// TIA Portal V15.1 export
// export: Created 2024-06-21T08:40:50.3190684Z, ExportSetting WithDefaults, DisplayName Totally Integrated Automation Portal, DisplayVersion V15.1 Update 5, DisplayName TIA Portal Openness, DisplayVersion V15.1 Update 5, DisplayName SINAMICS Startdrive Advanced, DisplayVersion V15.1, DisplayName G130, G150, S120, S150, SINAMICS MV, S210, DisplayVersion V15.1, DisplayName G110M, G120, G120C, G120D, G120P, DisplayVersion V15.1, DisplayName STEP 7 Professional, DisplayVersion V15.1 Update 5, DisplayName STEP 7 Safety, DisplayVersion V15.1, DisplayName WinCC Professional, DisplayVersion V15.1 Update 5, DisplayName SIMATIC Visualization Architect, DisplayVersion V15.1
DATA_BLOCK "_209230ZS01PNIODiag"   // DB424
{ S7_Optimized_Access := 'FALSE' }
AUTHOR : VCC
VERSION : 0.1
// stored: AutoNumber false, DBAccessibleFromOPCUA true, IsOnlyStoredInLoadMemory false, IsWriteProtectedInAS false
   VAR RETAIN
      "AA_209230AS10-JW60" { ExternalAccessible := 'False'; ExternalVisible := 'False'; ExternalWritable := 'False'} : Bool;   // Profinet device don't exist - ET200sp I/O - Busnode 230AS10 - node 60
      "AA_209230AX01-JW61" { ExternalAccessible := 'False'; ExternalVisible := 'False'; ExternalWritable := 'False'} : Bool;   // Profinet device don't exist - ET200sp I/O - Busnode 230AX01 - node 61
      "AB_209230CA21M4-UE150" { ExternalAccessible := 'False'; ExternalVisible := 'False'; ExternalWritable := 'False'} : Bool;   // Profinet device don't exist - MoviFit - 230CA21M4 - node 150
      "AB_209230CHB21M14-UE151" { ExternalAccessible := 'False'; ExternalVisible := 'False'; ExternalWritable := 'False'} : Bool;   // Profinet device don't exist - MoviFit - 230CHB21M14 - node 151
      "AB_209230CHB22M14-UE152" { ExternalAccessible := 'False'; ExternalVisible := 'False'; ExternalWritable := 'False'} : Bool;   // Profinet device don't exist - MoviFit - 230CHB22M14 - node 152
      "AB_209230CR22M1-UE153" { ExternalAccessible := 'False'; ExternalVisible := 'False'; ExternalWritable := 'False'} : Bool;   // Profinet device don't exist - MoviFit - 230CR22M1 - node 153
      "AA_209230ASD01-JW190" { ExternalAccessible := 'False'; ExternalVisible := 'False'; ExternalWritable := 'False'} : Bool;   // Profinet device don't exist - Euchner Door - 230ASD01 - node 190
      "AA_209230Field-JW223" { ExternalAccessible := 'False'; ExternalVisible := 'False'; ExternalWritable := 'False'} : Bool;   // Profinet device don't exist - Field Switch - Safety Zone 230 - node 223
      "AC_209230AS10-JW60Fault" { ExternalAccessible := 'False'; ExternalVisible := 'False'; ExternalWritable := 'False'} : Bool;   // Faulty profinet device -> For more detail information look for N.A. alarms in the alarmlist - ET200sp I/O - Busnode 230AS10 - node 60
      "AC_209230AX01-JW61Fault" { ExternalAccessible := 'False'; ExternalVisible := 'False'; ExternalWritable := 'False'} : Bool;   // Faulty profinet device -> For more detail information look for N.A. alarms in the alarmlist - ET200sp I/O - Busnode 230AX01 - node 61
      "AC_209230CA21M4-UE150Fault" { ExternalAccessible := 'False'; ExternalVisible := 'False'; ExternalWritable := 'False'} : Bool;   // Faulty profinet device -> For more detail information look for N.A. alarms in the alarmlist - MoviFit - 230CA21M4 - node 150
      "AC_209230CHB21M14-UE151Fault" { ExternalAccessible := 'False'; ExternalVisible := 'False'; ExternalWritable := 'False'} : Bool;   // Faulty profinet device -> For more detail information look for N.A. alarms in the alarmlist - MoviFit - 230CHB21M14 - node 151
      "AC_209230CHB22M14-UE152Fault" { ExternalAccessible := 'False'; ExternalVisible := 'False'; ExternalWritable := 'False'} : Bool;   // Faulty profinet device -> For more detail information look for N.A. alarms in the alarmlist - MoviFit - 230CHB22M14 - node 152
      "AC_209230CR22M1-UE153Fault" { ExternalAccessible := 'False'; ExternalVisible := 'False'; ExternalWritable := 'False'} : Bool;   // Faulty profinet device -> For more detail information look for N.A. alarms in the alarmlist - MoviFit - 230CR22M1 - node 153
      "AC_209230ASD01-JW190Fault" { ExternalAccessible := 'False'; ExternalVisible := 'False'; ExternalWritable := 'False'} : Bool;   // Faulty profinet device -> For more detail information look for N.A. alarms in the alarmlist - Euchner Door - 230ASD01 - node 190
      "AC_209230Field-JW223Fault" { ExternalAccessible := 'False'; ExternalVisible := 'False'; ExternalWritable := 'False'} : Bool;   // Faulty profinet device -> For more detail information look for N.A. alarms in the alarmlist - Field Switch - Safety Zone 230 - node 223
      "209230AS10-JW60AlarmABCondition" { ExternalAccessible := 'False'; ExternalVisible := 'False'; ExternalWritable := 'False'} : Bool;   // Alarm AB condition
      "209230AX01-JW61AlarmABCondition" { ExternalAccessible := 'False'; ExternalVisible := 'False'; ExternalWritable := 'False'} : Bool;   // Alarm AB condition
      "209230CA21M4-UE150AlarmABCondition" { ExternalAccessible := 'False'; ExternalVisible := 'False'; ExternalWritable := 'False'} : Bool;   // Alarm AB condition
      "209230CHB21M14-UE151AlarmABCondition" { ExternalAccessible := 'False'; ExternalVisible := 'False'; ExternalWritable := 'False'} : Bool;   // Alarm AB condition
      "209230CHB22M14-UE152AlarmABCondition" { ExternalAccessible := 'False'; ExternalVisible := 'False'; ExternalWritable := 'False'} : Bool;   // Alarm AB condition
      "209230CR22M1-UE153AlarmABCondition" { ExternalAccessible := 'False'; ExternalVisible := 'False'; ExternalWritable := 'False'} : Bool;   // Alarm AB condition
      "209230ASD01-JW190AlarmABCondition" { ExternalAccessible := 'False'; ExternalVisible := 'False'; ExternalWritable := 'False'} : Bool;   // Alarm AB condition
      "209230Field-JW223AlarmABCondition" { ExternalAccessible := 'False'; ExternalVisible := 'False'; ExternalWritable := 'False'} : Bool;   // Alarm AB condition
      "H_209230AS10-JW60IAnim" : Word;   // HMI Animation of the icon
      "H_209230AX01-JW61IAnim" : Word;   // HMI Animation of the icon
      "H_209230CA21M4-UE150IAnim" : Word;   // HMI Animation of the icon
      "H_209230CHB21M14-UE151IAnim" : Word;   // HMI Animation of the icon
      "H_209230CHB22M14-UE152IAnim" : Word;   // HMI Animation of the icon
      "H_209230CR22M1-UE153IAnim" : Word;   // HMI Animation of the icon
      "H_209230ASD01-JW190IAnim" : Word;   // HMI Animation of the icon
      "H_209230Field-JW223IAnim" : Word;   // HMI Animation of the icon
      "H_209230AS10-JW60IAnim2" : Word;   // HMI Animation of the icon
      "H_209230AX01-JW61IAnim2" : Word;   // HMI Animation of the icon
      "H_209230CA21M4-UE150IAnim2" : Word;   // HMI Animation of the icon
      "H_209230CHB21M14-UE151IAnim2" : Word;   // HMI Animation of the icon
      "H_209230CHB22M14-UE152IAnim2" : Word;   // HMI Animation of the icon
      "H_209230CR22M1-UE153IAnim2" : Word;   // HMI Animation of the icon
      "H_209230ASD01-JW190IAnim2" : Word;   // HMI Animation of the icon
      "H_209230Field-JW223IAnim2" : Word;   // HMI Animation of the icon
      H_IAnim : Word;   // Icon Animation / Animation
      H_Anim : Word;   // Animation
      H_DBnr : Int;   // DB number
      AlarmA { ExternalAccessible := 'False'; ExternalVisible := 'False'; ExternalWritable := 'False'} : Bool;   // Summary Alarm A
      AlarmB { ExternalAccessible := 'False'; ExternalVisible := 'False'; ExternalWritable := 'False'} : Bool;   // Summary Alarm B
      AlarmC { ExternalAccessible := 'False'; ExternalVisible := 'False'; ExternalWritable := 'False'} : Bool;   // Summary Alarm C
      AlarmD { ExternalAccessible := 'False'; ExternalVisible := 'False'; ExternalWritable := 'False'} : Bool;   // Summary Alarm D
      AlarmABCondition { ExternalAccessible := 'False'; ExternalVisible := 'False'; ExternalWritable := 'False'} : Bool;   // Alarm AB Condition
   END_VAR
BEGIN
END_DATA_BLOCK
